// TIA Portal project "elevador" (V16)
// Vorlageprojekt für das Buch mit Zielsystem S7-1200

(* hardware
DEVICE "S7-1200-Station_1"  S7-1200 Station
   slot 0: "Baugruppenträger_0"  Rack  V1.0
   slot 1: "PLC_1"  CPU 1211C DC/DC/DC  6ES7 211-1AE40-0XB0  V4.1
*)

// ===== PLC "PLC_1"  CPU 1211C DC/DC/DC =====

VAR_GLOBAL   // PLC tag table "Standard-Variablentabelle"
   "At elevator" AT %I0.3 : Bool;
   "At entry" AT %I0.4 : Bool;
   "At exit" AT %I0.5 : Bool;
   "At 0 (low)" AT %I0.6 : Bool;
   "At 0 (high)" AT %I0.7 : Bool;
   "At 1 (low)" AT %I1.0 : Bool;
   "At 1 (high)" AT %I1.1 : Bool;
   "At 2 (low)" AT %I1.2 : Bool;
   "At 2 (high)" AT %I1.3 : Bool;
   "At 3 (low)" AT %I1.4 : Bool;
   "At 3 (high)" AT %I1.5 : Bool;
   "Start" AT %I1.6 : Bool;
   "Reset" AT %I1.7 : Bool;
   "Stop" AT %I2.0 : Bool;
   "Emergency stop" AT %I2.1 : Bool;
   "Conveyor 0" AT %Q0.0 : Bool;
   "Conveyor 1" AT %Q0.1 : Bool;
   "Conveyor 2" AT %Q0.2 : Bool;
   "Conveyor 3" AT %Q0.3 : Bool;
   "Exit conveyor" AT %Q0.4 : Bool;
   "Load" AT %Q0.5 : Bool;
   "Unload" AT %Q0.6 : Bool;
   "Up" AT %Q0.7 : Bool;
   "Slow" AT %Q1.0 : Bool;
   "Down" AT %Q1.1 : Bool;
   "Warning light" AT %Q1.2 : Bool;
   "Start light" AT %Q1.3 : Bool;
   "Stop light" AT %Q1.5 : Bool;
   "Floor 1" AT %Q1.6 : Bool;
   "Floor 2" AT %Q1.7 : Bool;
   "Floor 3" AT %Q2.0 : Bool;
   "Position" AT %MW5 : Word;
END_VAR

// folder: System blocks/Program resources

DATA_BLOCK "IEC_Timer_0_DB"   // DB1
{ S7_Optimized_Access := 'TRUE' }
AUTHOR : Simatic
FAMILY : IEC
NAME : IEC_TMR
VERSION : 1.0
// stored: InstanceOfName IEC_TIMER
"IEC_TIMER"
BEGIN
END_DATA_BLOCK

DATA_BLOCK "IEC_Timer_0_DB_1"   // DB2
{ S7_Optimized_Access := 'TRUE' }
AUTHOR : Simatic
FAMILY : IEC
NAME : IEC_TMR
VERSION : 1.0
// stored: InstanceOfName IEC_TIMER
"IEC_TIMER"
BEGIN
END_DATA_BLOCK

DATA_BLOCK "IEC_Timer_0_DB_2"   // DB3
{ S7_Optimized_Access := 'TRUE' }
AUTHOR : Simatic
FAMILY : IEC
NAME : IEC_TMR
VERSION : 1.0
// stored: InstanceOfName IEC_TIMER
"IEC_TIMER"
BEGIN
END_DATA_BLOCK

DATA_BLOCK "IEC_Timer_0_DB_3"   // DB4
{ S7_Optimized_Access := 'TRUE' }
AUTHOR : Simatic
FAMILY : IEC
NAME : IEC_TMR
VERSION : 1.0
// stored: InstanceOfName IEC_TIMER
"IEC_TIMER"
BEGIN
END_DATA_BLOCK

DATA_BLOCK "IEC_Timer_0_DB_4"   // DB5
{ S7_Optimized_Access := 'TRUE' }
AUTHOR : Simatic
FAMILY : IEC
NAME : IEC_TMR
VERSION : 1.0
// stored: InstanceOfName IEC_TIMER
"IEC_TIMER"
BEGIN
END_DATA_BLOCK

DATA_BLOCK "IEC_Timer_0_DB_5"   // DB6
{ S7_Optimized_Access := 'TRUE' }
AUTHOR : Simatic
FAMILY : IEC
NAME : IEC_TMR
VERSION : 1.0
// stored: InstanceOfName IEC_TIMER
"IEC_TIMER"
BEGIN
END_DATA_BLOCK

// folder: (top level)

FUNCTION "MHJ-PLC-Lab-Function-S71200" : Void   // FC9000, SCL
{ S7_Optimized_Access := 'TRUE' }
VERSION : 0.1
   VAR_TEMP
      rdTimeReturn : Int;
      outputTime : DTL;
      SyncVal : Byte;
      forVal : Int;
      forVal_2 : Int;
      Value : Byte;
   END_VAR
   VAR CONSTANT
      CompVal : Byte := 16#34;
      Value_01 : Byte := 16#11;
      Value_01_DW : DWord := 16#A165_D992;
      Value_02_DW : DWord := 16#58BE_4401;
   END_VAR
BEGIN

   #Value:=PEEK(area := 16#82,
        dbNumber := 0,
        byteOffset := 511);
   #Value := #Value + 1;

   POKE(area := 16#82,
        dbNumber := 0,
        byteOffset := 511,
        value := #Value);

   POKE(area:=16#81,
        dbNumber:=0,
        byteOffset:=1016,
        value:=#Value_01_DW);
   POKE(area := 16#81,
        dbNumber := 0,
        byteOffset := 1020,
        value := #Value_02_DW);

   POKE(area := 16#81,
        dbNumber := 0,
        byteOffset := 511,
        value := B#16#00);

   FOR #forVal := 0 TO 120 DO
       FOR #forVal_2:=0 TO 10 DO
           #rdTimeReturn:=RD_SYS_T(#outputTime);
           #rdTimeReturn := WR_SYS_T(#outputTime);
           #rdTimeReturn := RD_SYS_T(#outputTime);
           #rdTimeReturn := WR_SYS_T(#outputTime);
       END_FOR;
       #SyncVal:= PEEK(area := 16#81,
                      dbNumber := 0,
                      byteOffset := 511);
       IF #SyncVal = #CompVal THEN
          GOTO M_1;
       END_IF;
   END_FOR;
   RETURN;

   M_1:
   POKE(area := 16#81,
        dbNumber := 0,
        byteOffset := 511,
        value := B#16#0);
END_FUNCTION

ORGANIZATION_BLOCK "Main"   // OB1, LAD, ProgramCycle
TITLE = "Main Program Sweep (Cycle)"
{ S7_Optimized_Access := 'TRUE' }
VERSION : 0.1
   VAR_INPUT
      Initial_Call : Bool;   // Initial call of this OB
      Remanence : Bool;   // =True, if remanent data are available
   END_VAR
   VAR_TEMP   // added for the SCL form of the ladder/FBD networks
      _w1 : Bool;
      _w2 : Bool;
      _w3 : Bool;
      _w4 : Bool;
   END_VAR
BEGIN

REGION Network 1: Konnektierungsbaustein für PLC-Lab
   // Im Netzwerk 1 wird der Konnektierungsbaustein für PLC-Lab aufgerufen.
   // Dieser Aufruf darf nicht entfernt werden!
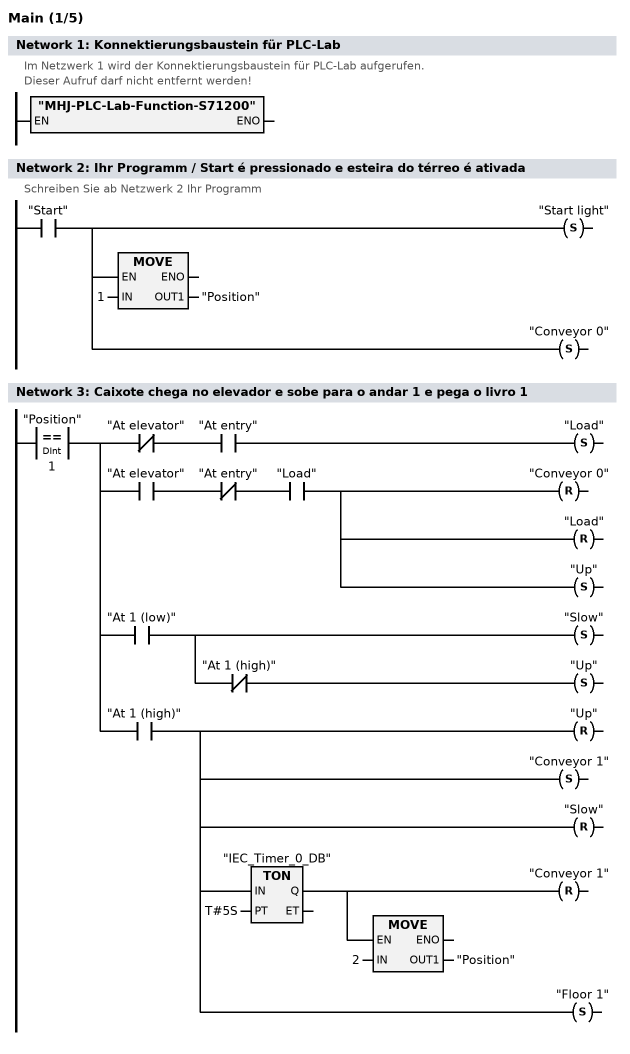
   RUNG wire#powerrail
      "MHJ-PLC-Lab-Function-S71200"()
   END_RUNG
   // the same network as SCL:
   "MHJ-PLC-Lab-Function-S71200"();
END_REGION

REGION Network 2: Ihr Programm / Start é pressionado e esteira do térreo é ativada
   // Schreiben Sie ab Netzwerk 2 Ihr Programm
   RUNG wire#powerrail
      Contact( "Start" )
      wire#w1
      S_Coil( "Start light" )
   END_RUNG
   RUNG wire#w1
      Move(in := 1, out1 => "Position")
   END_RUNG
   RUNG wire#w1
      S_Coil( "Conveyor 0" )
   END_RUNG
   // the same network as SCL:
   IF "Start" THEN
       "Start light" := TRUE;
       "Position" := 1;
       "Conveyor 0" := TRUE;
   END_IF;
END_REGION

REGION Network 3: Caixote chega no elevador e sobe para o andar 1 e pega o livro 1
   #_w1 := "Position" = 1;
   IF #_w1 AND NOT "At elevator" AND "At entry" THEN "Load" := TRUE; END_IF;
   IF #_w1 AND "At elevator" AND NOT "At entry" AND "Load" THEN "Conveyor 0" := FALSE; END_IF;
   #_w2 := #_w1 AND "At elevator" AND NOT "At entry" AND "Load";
   IF #_w2 THEN
       "Load" := FALSE;
       "Up" := TRUE;
   END_IF;
   #_w3 := #_w1 AND "At 1 (low)";
   IF #_w3 THEN "Slow" := TRUE; END_IF;
   IF #_w3 AND NOT "At 1 (high)" THEN "Up" := TRUE; END_IF;
   #_w4 := #_w1 AND "At 1 (high)";
   IF #_w4 THEN
       "Up" := FALSE;
       "Conveyor 1" := TRUE;
       "Slow" := FALSE;
   END_IF;
   "IEC_Timer_0_DB".TON(IN := #_w4, PT := T#5S);
   IF "IEC_Timer_0_DB".Q THEN
       "Conveyor 1" := FALSE;
       "Position" := 2;
   END_IF;
   IF #_w4 THEN "Floor 1" := TRUE; END_IF;
END_REGION

REGION Network 4: Caixote sobe para o andar 2 e pega o livro 2
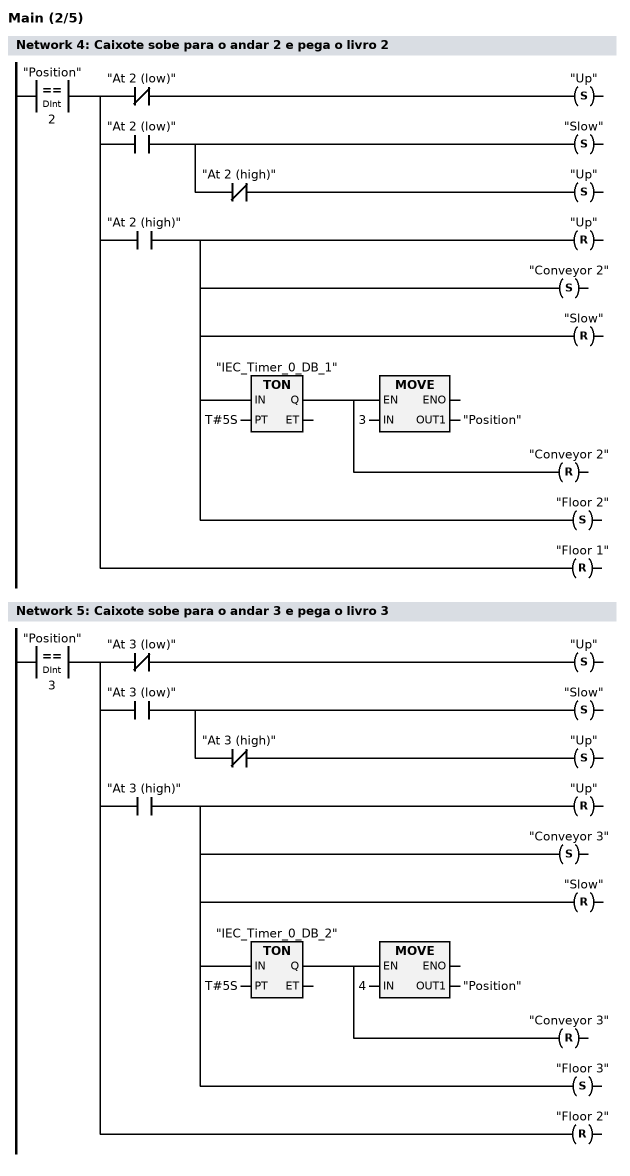
   #_w1 := "Position" = 2;
   IF #_w1 AND NOT "At 2 (low)" THEN "Up" := TRUE; END_IF;
   #_w2 := #_w1 AND "At 2 (low)";
   IF #_w2 THEN "Slow" := TRUE; END_IF;
   IF #_w2 AND NOT "At 2 (high)" THEN "Up" := TRUE; END_IF;
   #_w3 := #_w1 AND "At 2 (high)";
   IF #_w3 THEN
       "Up" := FALSE;
       "Conveyor 2" := TRUE;
       "Slow" := FALSE;
   END_IF;
   "IEC_Timer_0_DB_1".TON(IN := #_w3, PT := T#5S);
   IF "IEC_Timer_0_DB_1".Q THEN
       "Position" := 3;
       "Conveyor 2" := FALSE;
   END_IF;
   IF #_w3 THEN "Floor 2" := TRUE; END_IF;
   IF #_w1 THEN "Floor 1" := FALSE; END_IF;
END_REGION

REGION Network 5: Caixote sobe para o andar 3 e pega o livro 3
   #_w1 := "Position" = 3;
   IF #_w1 AND NOT "At 3 (low)" THEN "Up" := TRUE; END_IF;
   #_w2 := #_w1 AND "At 3 (low)";
   IF #_w2 THEN "Slow" := TRUE; END_IF;
   IF #_w2 AND NOT "At 3 (high)" THEN "Up" := TRUE; END_IF;
   #_w3 := #_w1 AND "At 3 (high)";
   IF #_w3 THEN
       "Up" := FALSE;
       "Conveyor 3" := TRUE;
       "Slow" := FALSE;
   END_IF;
   "IEC_Timer_0_DB_2".TON(IN := #_w3, PT := T#5S);
   IF "IEC_Timer_0_DB_2".Q THEN
       "Position" := 4;
       "Conveyor 3" := FALSE;
   END_IF;
   IF #_w3 THEN "Floor 3" := TRUE; END_IF;
   IF #_w1 THEN "Floor 2" := FALSE; END_IF;
END_REGION

REGION Network 6: Caixote desce para o andar 2 e pega o livro 4
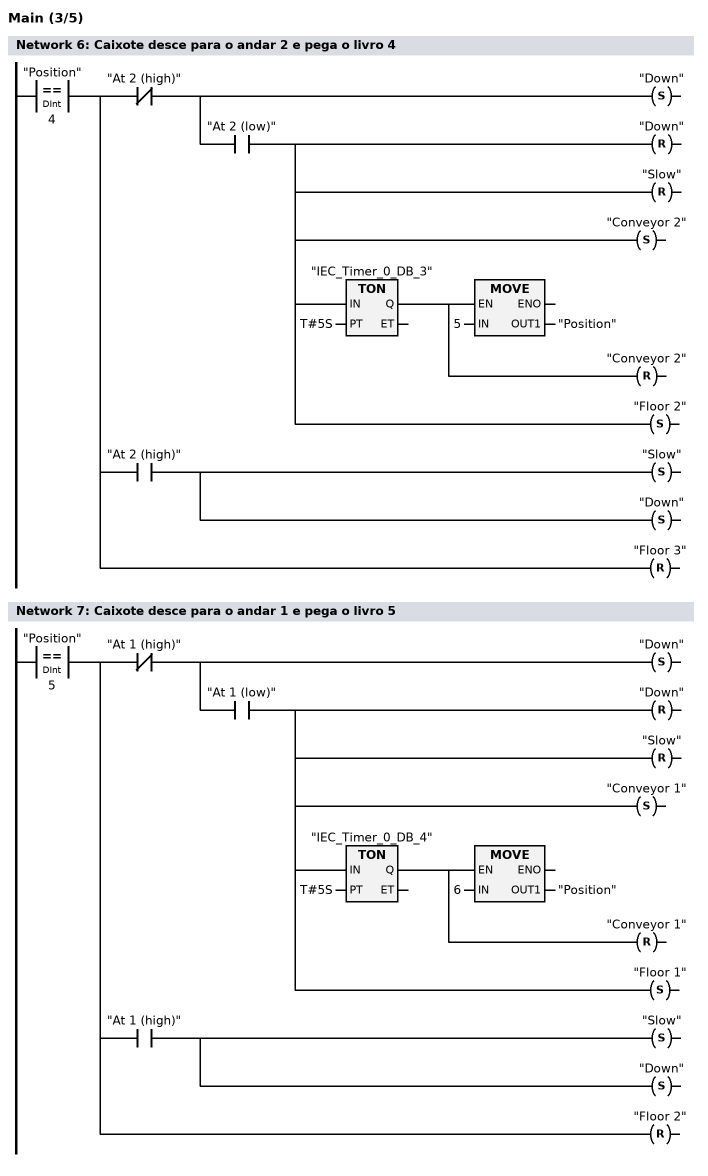
   #_w1 := "Position" = 4;
   #_w2 := #_w1 AND NOT "At 2 (high)";
   IF #_w2 THEN "Down" := TRUE; END_IF;
   #_w3 := #_w2 AND "At 2 (low)";
   IF #_w3 THEN
       "Down" := FALSE;
       "Slow" := FALSE;
       "Conveyor 2" := TRUE;
   END_IF;
   "IEC_Timer_0_DB_3".TON(IN := #_w3, PT := T#5S);
   IF "IEC_Timer_0_DB_3".Q THEN
       "Position" := 5;
       "Conveyor 2" := FALSE;
   END_IF;
   IF #_w3 THEN "Floor 2" := TRUE; END_IF;
   IF #_w1 AND "At 2 (high)" THEN
       "Slow" := TRUE;
       "Down" := TRUE;
   END_IF;
   IF #_w1 THEN "Floor 3" := FALSE; END_IF;
END_REGION

REGION Network 7: Caixote desce para o andar 1 e pega o livro 5
   #_w1 := "Position" = 5;
   #_w2 := #_w1 AND NOT "At 1 (high)";
   IF #_w2 THEN "Down" := TRUE; END_IF;
   #_w3 := #_w2 AND "At 1 (low)";
   IF #_w3 THEN
       "Down" := FALSE;
       "Slow" := FALSE;
       "Conveyor 1" := TRUE;
   END_IF;
   "IEC_Timer_0_DB_4".TON(IN := #_w3, PT := T#5S);
   IF "IEC_Timer_0_DB_4".Q THEN
       "Position" := 6;
       "Conveyor 1" := FALSE;
   END_IF;
   IF #_w3 THEN "Floor 1" := TRUE; END_IF;
   IF #_w1 AND "At 1 (high)" THEN
       "Slow" := TRUE;
       "Down" := TRUE;
   END_IF;
   IF #_w1 THEN "Floor 2" := FALSE; END_IF;
END_REGION

REGION Network 8: Caixote desce para o térreo para ser entregue
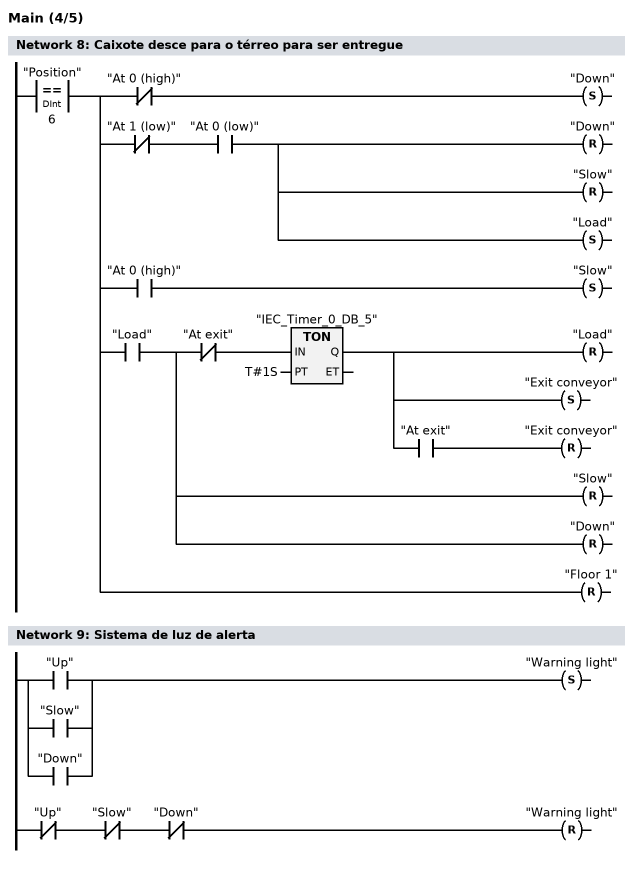
   #_w1 := "Position" = 6;
   IF #_w1 AND NOT "At 0 (high)" THEN "Down" := TRUE; END_IF;
   IF #_w1 AND NOT "At 1 (low)" AND "At 0 (low)" THEN
       "Down" := FALSE;
       "Slow" := FALSE;
       "Load" := TRUE;
   END_IF;
   IF #_w1 AND "At 0 (high)" THEN "Slow" := TRUE; END_IF;
   #_w2 := #_w1 AND "Load";
   "IEC_Timer_0_DB_5".TON(IN := #_w2 AND NOT "At exit", PT := T#1S);
   IF "IEC_Timer_0_DB_5".Q THEN
       "Load" := FALSE;
       "Exit conveyor" := TRUE;
   END_IF;
   IF "IEC_Timer_0_DB_5".Q AND "At exit" THEN "Exit conveyor" := FALSE; END_IF;
   IF #_w2 THEN
       "Slow" := FALSE;
       "Down" := FALSE;
   END_IF;
   IF #_w1 THEN "Floor 1" := FALSE; END_IF;
END_REGION

REGION Network 9: Sistema de luz de alerta
   RUNG wire#powerrail
      Contact( "Up" )
      wire#w1
      S_Coil( "Warning light" )
   END_RUNG
   RUNG wire#powerrail
      Contact( "Slow" )
   END_RUNG wire#w1
   RUNG wire#powerrail
      Contact( "Down" )
   END_RUNG wire#w1
   RUNG wire#powerrail
      I_Contact( "Up" )
      I_Contact( "Slow" )
      I_Contact( "Down" )
      R_Coil( "Warning light" )
   END_RUNG
   // the same network as SCL:
   IF "Up" OR "Slow" OR "Down" THEN "Warning light" := TRUE; END_IF;
   IF NOT "Up" AND NOT "Slow" AND NOT "Down" THEN "Warning light" := FALSE; END_IF;
END_REGION

REGION Network 10: Botão de pare e emergência
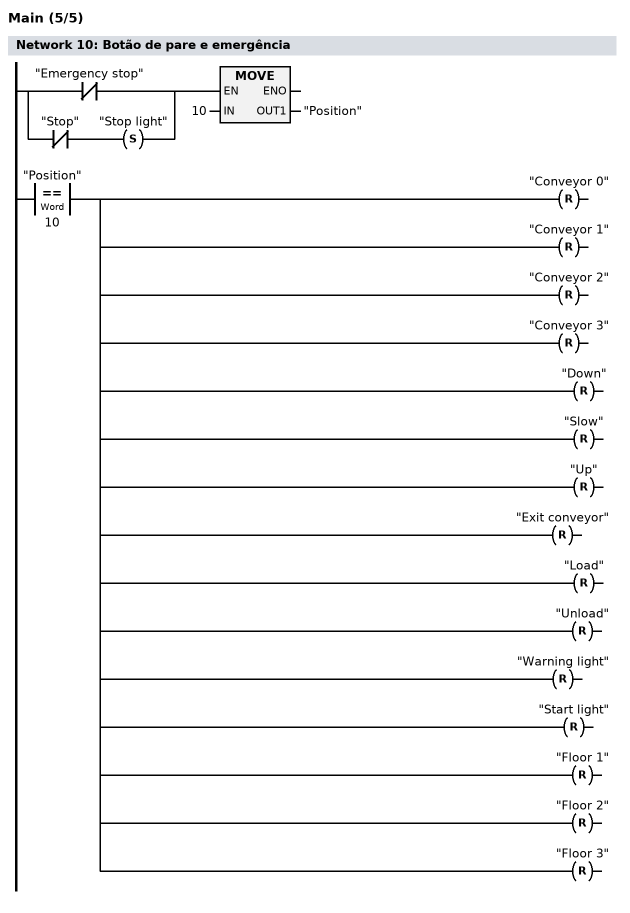
   RUNG wire#powerrail
      I_Contact( "Emergency stop" )
      wire#w1
      Move(in := 10, out1 => "Position")
   END_RUNG
   RUNG wire#powerrail
      I_Contact( "Stop" )
      S_Coil( "Stop light" )
   END_RUNG wire#w1
   RUNG wire#powerrail
      { S7_Templates := "SrcType := Word" } EQ_Contact(in1 := "Position", in2 := 10)
      wire#w2
      R_Coil( "Conveyor 0" )
   END_RUNG
   RUNG wire#w2
      R_Coil( "Conveyor 1" )
   END_RUNG
   RUNG wire#w2
      R_Coil( "Conveyor 2" )
   END_RUNG
   RUNG wire#w2
      R_Coil( "Conveyor 3" )
   END_RUNG
   RUNG wire#w2
      R_Coil( "Down" )
   END_RUNG
   RUNG wire#w2
      R_Coil( "Slow" )
   END_RUNG
   RUNG wire#w2
      R_Coil( "Up" )
   END_RUNG
   RUNG wire#w2
      R_Coil( "Exit conveyor" )
   END_RUNG
   RUNG wire#w2
      R_Coil( "Load" )
   END_RUNG
   RUNG wire#w2
      R_Coil( "Unload" )
   END_RUNG
   RUNG wire#w2
      R_Coil( "Warning light" )
   END_RUNG
   RUNG wire#w2
      R_Coil( "Start light" )
   END_RUNG
   RUNG wire#w2
      R_Coil( "Floor 1" )
   END_RUNG
   RUNG wire#w2
      R_Coil( "Floor 2" )
   END_RUNG
   RUNG wire#w2
      R_Coil( "Floor 3" )
   END_RUNG
   // the same network as SCL:
   IF NOT "Stop" THEN "Stop light" := TRUE; END_IF;
   IF NOT "Emergency stop" OR NOT "Stop" THEN "Position" := 10; END_IF;
   IF "Position" = 10 THEN
       "Conveyor 0" := FALSE;
       "Conveyor 1" := FALSE;
       "Conveyor 2" := FALSE;
       "Conveyor 3" := FALSE;
       "Down" := FALSE;
       "Slow" := FALSE;
       "Up" := FALSE;
       "Exit conveyor" := FALSE;
       "Load" := FALSE;
       "Unload" := FALSE;
       "Warning light" := FALSE;
       "Start light" := FALSE;
       "Floor 1" := FALSE;
       "Floor 2" := FALSE;
       "Floor 3" := FALSE;
   END_IF;
END_REGION
END_ORGANIZATION_BLOCK